Staubli VAL3: onF8Event.pgx

program onF8Event()
  local string l_sMessage
begin
  // look if the bButton is enable
  if bButton[7]
    //
    //
    // TERMINATE CYCLE
    //
    if cycleStatus:bCycle and !cycleStatus:bEnding
      logMsg("[KERNEL] INTERFACE:End cycle")
      //
      cycleStatus:bToEnd=true
      call language:message(l_sMessage,3)
      popUpMsg(l_sMessage)
    endIf
  endIf
end
